// TIA Portal V17 export
// export: Created 2024-08-07T21:44:00.7551322Z, ExportSetting WithDefaults, DisplayName Totally Integrated Automation Portal, DisplayVersion V17 Update 7, DisplayName TIA Portal Openness, DisplayVersion V17 Update 7, DisplayName TIA Portal Version Control Interface, DisplayVersion V17, DisplayName SINAMICS Startdrive Advanced, DisplayVersion V17 SP2, DisplayName SINAMICS Startdrive G110M, G120, G120C, G120D, G120P, G115D, DisplayVersion V17 SP2, DisplayName SINAMICS Startdrive G130, G150, S120, S150, SINAMICS MV, S210, DisplayVersion V17 SP2, DisplayName STEP 7 Professional, DisplayVersion V17 Update 7, DisplayName STEP 7 Safety, DisplayVersion V17 Update 6, DisplayName WinCC Advanced / Unified PC, DisplayVersion V17 Update 7
ORGANIZATION_BLOCK "OB_ProgramCycle"   // OB1, LAD, ProgramCycle
TITLE = "Main Program Sweep (Cycle)"
{ S7_Optimized_Access := 'TRUE' }
VERSION : 0.1
// stored: AutoNumber true, IsIECCheckEnabled false, SetENOAutomatically false
   VAR_INPUT
      Initial_Call : Bool;   // Initial call of this OB
      Remanence : Bool;   // =True, if remanent data are available
   END_VAR
   VAR_TEMP   // added for the SCL form of the ladder/FBD networks
      _w1 : Bool;
      _s5time1 : S5Time;
   END_VAR
BEGIN

REGION Network 1
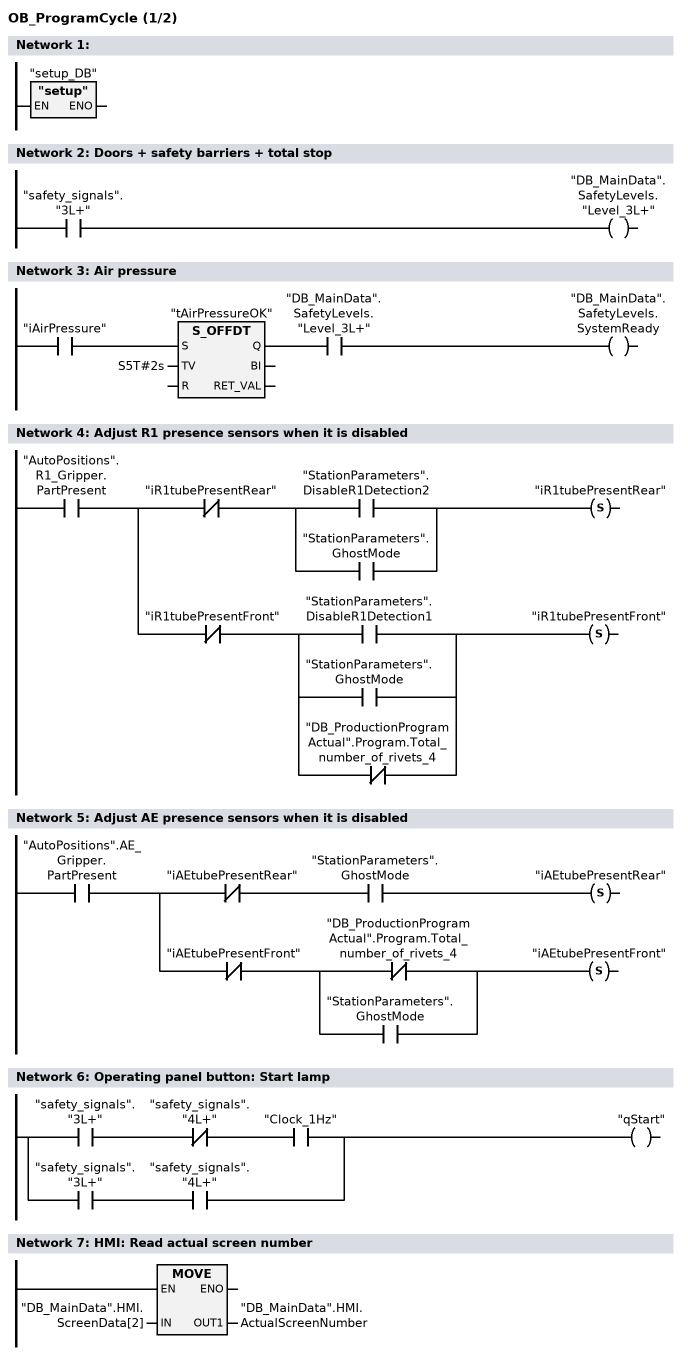
   RUNG wire#powerrail
      "setup_DB"()
   END_RUNG
   // the same network as SCL:
   "setup_DB"();   // "setup"
END_REGION

REGION Network 2: Doors + safety barriers + total stop
   RUNG wire#powerrail
      Contact( "safety_signals"."3L+" )
      Coil( "DB_MainData".SafetyLevels."Level_3L+" )
   END_RUNG
   // the same network as SCL:
   "DB_MainData".SafetyLevels."Level_3L+" := "safety_signals"."3L+";
END_REGION

REGION Network 3: Air pressure
   RUNG wire#powerrail
      Contact( "iAirPressure" )
      S_OFFDT(T_NO := "tAirPressureOK", TV := S5T#2s, R :=, BI =>, RET_VAL =>)
      Contact( "DB_MainData".SafetyLevels."Level_3L+" )
      Coil( "DB_MainData".SafetyLevels.SystemReady )
   END_RUNG
   // the same network as SCL:
   #_s5time1 := S_OFFDT(T_NO := "tAirPressureOK", S := "iAirPressure", TV := S5T#2s, Q => #_w1);
   "DB_MainData".SafetyLevels.SystemReady := #_w1 AND "DB_MainData".SafetyLevels."Level_3L+";
END_REGION

REGION Network 4: Adjust R1 presence sensors when it is disabled
   RUNG wire#powerrail
      Contact( "AutoPositions".R1_Gripper.PartPresent )
      wire#w1
      I_Contact( "iR1tubePresentRear" )
      wire#w2
      Contact( "StationParameters".DisableR1Detection2 )
      wire#w3
      S_Coil( "iR1tubePresentRear" )
   END_RUNG
   RUNG wire#w2
      Contact( "StationParameters".GhostMode )
   END_RUNG wire#w3
   RUNG wire#w1
      I_Contact( "iR1tubePresentFront" )
      wire#w4
      Contact( "StationParameters".DisableR1Detection1 )
      wire#w5
      S_Coil( "iR1tubePresentFront" )
   END_RUNG
   RUNG wire#w4
      Contact( "StationParameters".GhostMode )
   END_RUNG wire#w5
   RUNG wire#w4
      I_Contact( "DB_ProductionProgramActual".Program.Total_number_of_rivets_4 )
   END_RUNG wire#w5
   // the same network as SCL:
   IF "AutoPositions".R1_Gripper.PartPresent AND NOT "iR1tubePresentRear" AND ("StationParameters".DisableR1Detection2 OR "StationParameters".GhostMode) THEN
       "iR1tubePresentRear" := TRUE;
   END_IF;
   IF "AutoPositions".R1_Gripper.PartPresent AND NOT "iR1tubePresentFront" AND ("StationParameters".DisableR1Detection1 OR "StationParameters".GhostMode OR NOT "DB_ProductionProgramActual".Program.Total_number_of_rivets_4) THEN
       "iR1tubePresentFront" := TRUE;
   END_IF;
END_REGION

REGION Network 5: Adjust AE presence sensors when it is disabled
   RUNG wire#powerrail
      Contact( "AutoPositions".AE_Gripper.PartPresent )
      wire#w1
      I_Contact( "iAEtubePresentRear" )
      Contact( "StationParameters".GhostMode )
      S_Coil( "iAEtubePresentRear" )
   END_RUNG
   RUNG wire#w1
      I_Contact( "iAEtubePresentFront" )
      wire#w2
      I_Contact( "DB_ProductionProgramActual".Program.Total_number_of_rivets_4 )
      wire#w3
      S_Coil( "iAEtubePresentFront" )
   END_RUNG
   RUNG wire#w2
      Contact( "StationParameters".GhostMode )
   END_RUNG wire#w3
   // the same network as SCL:
   IF "AutoPositions".AE_Gripper.PartPresent AND NOT "iAEtubePresentRear" AND "StationParameters".GhostMode THEN
       "iAEtubePresentRear" := TRUE;
   END_IF;
   IF "AutoPositions".AE_Gripper.PartPresent AND NOT "iAEtubePresentFront" AND (NOT "DB_ProductionProgramActual".Program.Total_number_of_rivets_4 OR "StationParameters".GhostMode) THEN
       "iAEtubePresentFront" := TRUE;
   END_IF;
END_REGION

REGION Network 6: Operating panel button: Start lamp
   RUNG wire#powerrail
      Contact( "safety_signals"."3L+" )
      I_Contact( "safety_signals"."4L+" )
      Contact( "Clock_1Hz" )
      wire#w1
      Coil( "qStart" )
   END_RUNG
   RUNG wire#powerrail
      Contact( "safety_signals"."3L+" )
      Contact( "safety_signals"."4L+" )
   END_RUNG wire#w1
   // the same network as SCL:
   "qStart" := ("safety_signals"."3L+" AND NOT "safety_signals"."4L+" AND "Clock_1Hz") OR ("safety_signals"."3L+" AND "safety_signals"."4L+");
END_REGION

REGION Network 7: HMI: Read actual screen number
   RUNG wire#powerrail
      Move(in := "DB_MainData".HMI.ScreenData[2], out1 => "DB_MainData".HMI.ActualScreenNumber)
   END_RUNG
   // the same network as SCL:
   "DB_MainData".HMI.ActualScreenNumber := "DB_MainData".HMI.ScreenData[2];
END_REGION

REGION Network 8: FB_Main
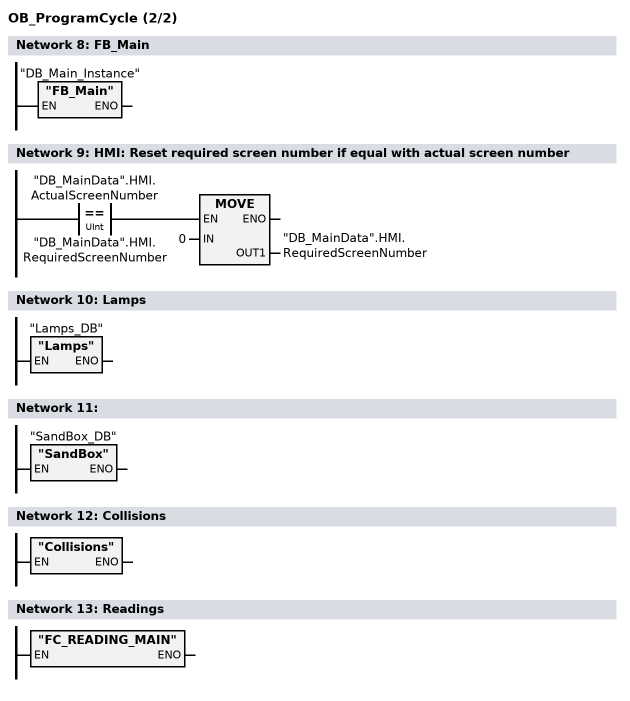
   RUNG wire#powerrail
      "DB_Main_Instance"()
   END_RUNG
   // the same network as SCL:
   "DB_Main_Instance"();   // "FB_Main"
END_REGION

REGION Network 9: HMI: Reset required screen number if equal with actual screen number
   RUNG wire#powerrail
      { S7_Templates := "SrcType := UInt" } EQ_Contact(in1 := "DB_MainData".HMI.ActualScreenNumber, in2 := "DB_MainData".HMI.RequiredScreenNumber)
      Move(in := 0, out1 => "DB_MainData".HMI.RequiredScreenNumber)
   END_RUNG
   // the same network as SCL:
   IF "DB_MainData".HMI.ActualScreenNumber = "DB_MainData".HMI.RequiredScreenNumber THEN
       "DB_MainData".HMI.RequiredScreenNumber := 0;
   END_IF;
END_REGION

REGION Network 10: Lamps
   RUNG wire#powerrail
      "Lamps_DB"()
   END_RUNG
   // the same network as SCL:
   "Lamps_DB"();   // "Lamps"
END_REGION

REGION Network 11
   RUNG wire#powerrail
      "SandBox_DB"()
   END_RUNG
   // the same network as SCL:
   "SandBox_DB"();   // "SandBox"
END_REGION

REGION Network 12: Collisions
   RUNG wire#powerrail
      "Collisions"()
   END_RUNG
   // the same network as SCL:
   "Collisions"();
END_REGION

REGION Network 13: Readings
   RUNG wire#powerrail
      "FC_READING_MAIN"()
   END_RUNG
   // the same network as SCL:
   "FC_READING_MAIN"();
END_REGION
END_ORGANIZATION_BLOCK
